Fanuc KAREL source: IO_MOD_TYPE.kl

PROGRAM T
%NOLOCKGROUP
VAR
 v0 : INTEGER
 v1 : INTEGER
 v2 : INTEGER
 v3 : INTEGER
BEGIN
 IO_MOD_TYPE(v0, v1, v2, v3)
END T
